PROGRAM P_WritePersistentData
VAR
	fbWritePersistentData: FB_WritePersistentData;
	StartTON: TON;
	iCounter: INT;

END_VAR

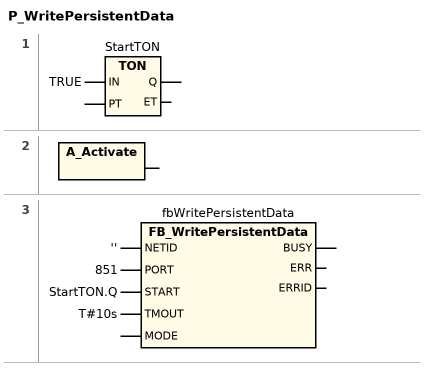
// NETWORK 1
StartTON(IN := TRUE); // TON

// NETWORK 2
A_Activate();

// NETWORK 3
fbWritePersistentData(NETID := '', PORT := 851, START := StartTON.Q, TMOUT := T#10s); // FB_WritePersistentData

ACTION A_Activate:

IF StartTON.Q THEN
	StartTON(IN := FALSE, PT:= T#1M);
		IF NOT fbWritePersistentData.BUSY THEN
		StartTON(IN := TRUE);
		iCounter := iCounter +1; IF iCounter > 50 THEN iCounter := 0; END_IF
		END_IF
END_IF
END_ACTION

END_PROGRAM

(* stored: Version 1.1.0.1, ProductVersion 3.1.4024.10
   POU P_WritePersistentData: Id {9273163e-f78f-4510-b2b7-6a9596e29f16}, SpecialFunc None
   Action A_Activate: Id {0ed701fc-d5d8-46b0-8d9d-38500e2fb304} *)
